TEXTLIST Txt_GridTypeSelection
  0 = 'Default'
  1 = 'Test_DyStartMark'
  2 = 'Test_AllDxFactor'
  3 = 'Test_AllDyFactor'
  4 = 'Test_DxColFactor'
  5 = 'Test_DyColFactro'
  6 = 'Test_Dx_FirstRowOnlyFactor'
   = ''
END_TEXTLIST

(* stored: Version 1.1.0.1, ProductVersion 3.1.4024.11
   TextList Txt_GridTypeSelection: Id {dfced12c-aca0-42b6-9fdc-4245b6e92103} *)
